ABB RAPID module: Module1.mod

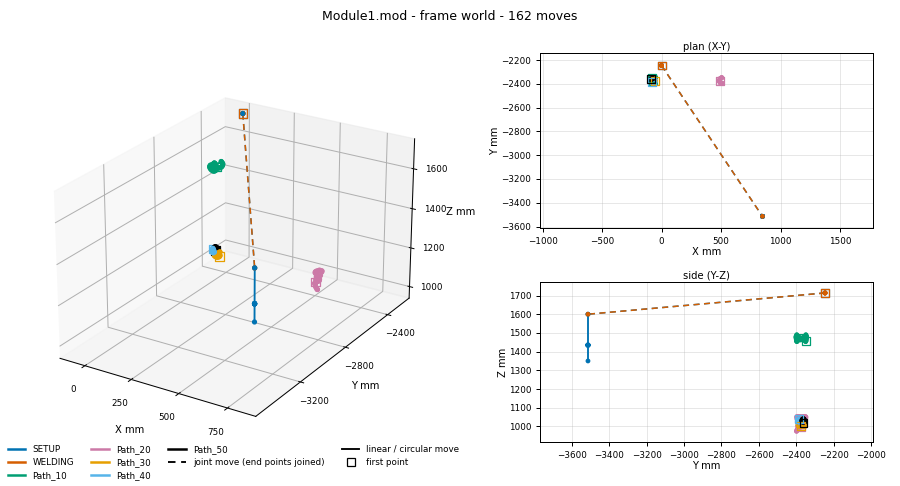
[picture p0: tool path of Module1.mod in frame world, 162 of 162 moves have a stored position in this frame; points joined in program order, loops and branches not executed]
MODULE Module1
    CONST robtarget Target_00:=[[0,-2246.385527781,1713.738524269],[0.23021145,-0.668582596,0.668582596,0.23021145],[0,0,0,0],[9E+09,9E+09,9E+09,9E+09,9E+09,9E+09]];
    CONST robtarget Target_10:=[[-80.421946623,-2349.93093018,1456.191919268],[0.23021145,-0.668582596,0.668582596,0.23021145],[0,0,0,0],[9E+09,9E+09,9E+09,9E+09,9E+09,9E+09]];
    CONST robtarget Target_20:=[[-85.308425352,-2349.8292418,1459.188833121],[0.23021145,-0.668582596,0.668582596,0.23021145],[0,0,0,0],[9E+09,9E+09,9E+09,9E+09,9E+09,9E+09]];
    CONST robtarget Target_30:=[[-89.179888675,-2349.715135272,1463.416236431],[0.23021145,-0.668582596,0.668582596,0.23021145],[0,0,0,0],[9E+09,9E+09,9E+09,9E+09,9E+09,9E+09]];
    CONST robtarget Target_40:=[[-91.78885584,-2349.595757829,1468.705305741],[0.23021145,-0.668582596,0.668582596,0.23021145],[0,0,0,0],[9E+09,9E+09,9E+09,9E+09,9E+09,9E+09]];
    CONST robtarget Target_50:=[[-92.546420184,-2350.235564494,1471.857704903],[0.23021145,-0.668582596,0.668582596,0.23021145],[0,0,0,0],[9E+09,9E+09,9E+09,9E+09,9E+09,9E+09]];
    CONST robtarget Target_60:=[[-92.795669653,-2352.001572523,1474.657635747],[0.23021145,-0.668582596,0.668582596,0.23021145],[0,0,0,0],[9E+09,9E+09,9E+09,9E+09,9E+09,9E+09]];
    CONST robtarget Target_70:=[[-92.744993461,-2354.535100522,1476.584408087],[0.23021145,-0.668582596,0.668582596,0.23021145],[0,0,0,0],[9E+09,9E+09,9E+09,9E+09,9E+09,9E+09]];
    CONST robtarget Target_80:=[[-92.678630412,-2357.601626995,1477.312867316],[0.23021145,-0.668582596,0.668582596,0.23021145],[0,0,0,0],[9E+09,9E+09,9E+09,9E+09,9E+09,9E+09]];
    CONST robtarget Target_10_3:=[[847.938,-3513.969,1435],[0.130526192,0,-0.991444861,0],[-1,0,0,0],[9E+09,9E+09,9E+09,9E+09,9E+09,9E+09]];
    CONST robtarget Target_10_4:=[[847.938,-3513.969,1435],[0.130526192,0,0.991444861,0],[-1,-1,0,0],[9E+09,9E+09,9E+09,9E+09,9E+09,9E+09]];
    CONST robtarget Target_10_2:=[[847.938,-3513.969,1435],[0,0,1,0],[0,-1,0,0],[9E+09,9E+09,9E+09,9E+09,9E+09,9E+09]];
    CONST robtarget Target_10_5:=[[847.938,-3513.969,1435],[0,0,0.991444861,-0.130526192],[-1,-1,0,0],[9E+09,9E+09,9E+09,9E+09,9E+09,9E+09]];
    CONST robtarget Target_10_6:=[[847.938,-3513.969,1435],[0,0,0.991444861,0.130526192],[-2,0,-1,0],[9E+09,9E+09,9E+09,9E+09,9E+09,9E+09]];
    CONST robtarget Target_10_7:=[[847.938,-3513.969,1350],[0,0,1,0],[-1,-1,0,0],[9E+09,9E+09,9E+09,9E+09,9E+09,9E+09]];
    CONST robtarget HOME:=[[0,-2246.385527781,1713.738524269],[0.23021145,-0.668582596,0.668582596,0.23021145],[0,-1,0,0],[9E+09,9E+09,9E+09,9E+09,9E+09,9E+09]];
    CONST robtarget SetUp0:=[[847.938,-3513.969,1600],[0,0,1,0],[0,-1,0,0],[9E+09,9E+09,9E+09,9E+09,9E+09,9E+09]];
    CONST robtarget SetUp1:=[[847.938,-3513.969,1435],[0,0,1,0],[0,-1,0,0],[9E+09,9E+09,9E+09,9E+09,9E+09,9E+09]];
    CONST robtarget SetUp_D:=[[847.938,-3513.969,1435],[0.130526192,0,-0.991444861,0],[-1,0,0,0],[9E+09,9E+09,9E+09,9E+09,9E+09,9E+09]];
    CONST robtarget SetUp_U:=[[847.938,-3513.969,1435],[0.130526192,0,0.991444861,0],[-1,-1,0,0],[9E+09,9E+09,9E+09,9E+09,9E+09,9E+09]];
    CONST robtarget SetUp_L:=[[847.938,-3513.969,1435],[0,0,0.991444861,-0.130526192],[-1,-1,0,0],[9E+09,9E+09,9E+09,9E+09,9E+09,9E+09]];
    CONST robtarget SetUp_R:=[[847.938,-3513.969,1435],[0,0,0.991444861,0.130526192],[-2,0,-1,0],[9E+09,9E+09,9E+09,9E+09,9E+09,9E+09]];
    CONST robtarget SetUp2:=[[847.938,-3513.969,1350],[0,0,1,0],[-1,-1,0,0],[9E+09,9E+09,9E+09,9E+09,9E+09,9E+09]];
    CONST robtarget Target_12:=[[-51.6,-2395.953,1475.08],[0.23021145,-0.668582596,0.668582596,0.23021145],[0,-1,0,0],[9E+09,9E+09,9E+09,9E+09,9E+09,9E+09]];
    CONST robtarget Target_11:=[[-76.443538654,-2395.952996748,1454.921874665],[0.23021145,-0.668582596,0.668582596,0.23021145],[0,-1,0,0],[9E+09,9E+09,9E+09,9E+09,9E+09,9E+09]];
    CONST robtarget Target_13:=[[-58.133756044,-2397.268954021,1490.12991755],[0.23021145,-0.668582596,0.668582596,0.23021145],[0,-1,0,0],[9E+09,9E+09,9E+09,9E+09,9E+09,9E+09]];
    CONST robtarget Target_14:=[[-58.130333404,-2349.245966493,1490.126743663],[0.23021145,-0.668582596,0.668582596,0.23021145],[0,-1,0,0],[9E+09,9E+09,9E+09,9E+09,9E+09,9E+09]];
    CONST robtarget Target_24:=[[-76.443540019,-2395.952934877,1454.921816349],[0.23021145,-0.668582596,0.668582596,0.23021145],[0,0,0,0],[9E+09,9E+09,9E+09,9E+09,9E+09,9E+09]];
    CONST robtarget Target_34:=[[-72.197140196,-2396.852775521,1454.480000199],[0.23021145,-0.668582596,0.668582596,0.23021145],[0,0,0,0],[9E+09,9E+09,9E+09,9E+09,9E+09,9E+09]];
    CONST robtarget Target_44:=[[-68.822373268,-2397.251160157,1454.75878848],[0.23021145,-0.668582596,0.668582596,0.23021145],[0,0,0,0],[9E+09,9E+09,9E+09,9E+09,9E+09,9E+09]];
    CONST robtarget Target_54:=[[-63.419325441,-2398.041235042,1456.445093127],[0.23021145,-0.668582596,0.668582596,0.23021145],[0,0,0,0],[9E+09,9E+09,9E+09,9E+09,9E+09,9E+09]];
    CONST robtarget Target_64:=[[-56.852171112,-2399.35121885,1461.339397818],[0.23021145,-0.668582596,0.668582596,0.23021145],[0,0,0,0],[9E+09,9E+09,9E+09,9E+09,9E+09,9E+09]];
    CONST robtarget Target_74:=[[-52.904973041,-2400.580201887,1467.86460433],[0.23021145,-0.668582596,0.668582596,0.23021145],[0,0,0,0],[9E+09,9E+09,9E+09,9E+09,9E+09,9E+09]];
    CONST robtarget Target_84:=[[-51.602040443,-2401.574973711,1474.790065418],[0.23021145,-0.668582596,0.668582596,0.23021145],[0,0,0,0],[9E+09,9E+09,9E+09,9E+09,9E+09,9E+09]];
    CONST robtarget Target_94:=[[-51.753594032,-2401.880985924,1477.590872953],[0.23021145,-0.668582596,0.668582596,0.23021145],[0,0,0,0],[9E+09,9E+09,9E+09,9E+09,9E+09,9E+09]];
    CONST robtarget Target_104:=[[-52.921425627,-2401.219597479,1482.339240328],[0.23021145,-0.668582596,0.668582596,0.23021145],[0,0,0,0],[9E+09,9E+09,9E+09,9E+09,9E+09,9E+09]];
    CONST robtarget Target_114:=[[-56.936344557,-2398.168943835,1488.914045775],[0.23021145,-0.668582596,0.668582596,0.23021145],[0,0,0,0],[9E+09,9E+09,9E+09,9E+09,9E+09,9E+09]];
    CONST robtarget Target_124:=[[-58.13387415,-2397.086440024,1490.130053275],[0.23021145,-0.668582596,0.668582596,0.23021145],[0,0,0,0],[9E+09,9E+09,9E+09,9E+09,9E+09,9E+09]];
    CONST robtarget Target_134:=[[-58.085063514,-2349.180158559,1490.084284988],[0.23021145,-0.668582596,0.668582596,0.23021145],[0,0,0,0],[9E+09,9E+09,9E+09,9E+09,9E+09,9E+09]];
    CONST robtarget Target_144:=[[-56.934648376,-2348.363913463,1488.91217408],[0.23021145,-0.668582596,0.668582596,0.23021145],[0,0,0,0],[9E+09,9E+09,9E+09,9E+09,9E+09,9E+09]];
    CONST robtarget Target_154:=[[-52.920814209,-2345.314117052,1482.337616361],[0.23021145,-0.668582596,0.668582596,0.23021145],[0,0,0,0],[9E+09,9E+09,9E+09,9E+09,9E+09,9E+09]];
    CONST robtarget Target_164:=[[-51.75346743,-2344.653327795,1477.589841799],[0.23021145,-0.668582596,0.668582596,0.23021145],[0,0,0,0],[9E+09,9E+09,9E+09,9E+09,9E+09,9E+09]];
    CONST robtarget Target_174:=[[-51.602106701,-2344.95991739,1474.785395815],[0.23021145,-0.668582596,0.668582596,0.23021145],[0,0,0,0],[9E+09,9E+09,9E+09,9E+09,9E+09,9E+09]];
    CONST robtarget Target_184:=[[-52.906744673,-2345.954949784,1467.859868499],[0.23021145,-0.668582596,0.668582596,0.23021145],[0,0,0,0],[9E+09,9E+09,9E+09,9E+09,9E+09,9E+09]];
    CONST robtarget Target_194:=[[-56.855846082,-2347.184083727,1461.335294093],[0.23021145,-0.668582596,0.668582596,0.23021145],[0,0,0,0],[9E+09,9E+09,9E+09,9E+09,9E+09,9E+09]];
    CONST robtarget Target_204:=[[-63.424235174,-2348.493945291,1456.442780476],[0.23021145,-0.668582596,0.668582596,0.23021145],[0,0,0,0],[9E+09,9E+09,9E+09,9E+09,9E+09,9E+09]];
    CONST robtarget Target_214:=[[-68.825579531,-2349.283560155,1454.75825582],[0.23021145,-0.668582596,0.668582596,0.23021145],[0,0,0,0],[9E+09,9E+09,9E+09,9E+09,9E+09,9E+09]];
    CONST robtarget Target_224:=[[-72.19902246,-2349.681691113,1454.480000023],[0.23021145,-0.668582596,0.668582596,0.23021145],[0,0,0,0],[9E+09,9E+09,9E+09,9E+09,9E+09,9E+09]];
    CONST robtarget Target_234:=[[-76.44321562,-2350.581156993,1454.921748062],[0.23021145,-0.668582596,0.668582596,0.23021145],[0,0,0,0],[9E+09,9E+09,9E+09,9E+09,9E+09,9E+09]];
    CONST robtarget Target_90:=[[-92.744993461,-2360.668153479,1476.584408087],[0.23021145,-0.668582596,0.668582596,0.23021145],[0,0,0,0],[9E+09,9E+09,9E+09,9E+09,9E+09,9E+09]];
    CONST robtarget Target_100:=[[-92.795669653,-2363.201681499,1474.657635755],[0.23021145,-0.668582596,0.668582596,0.23021145],[0,0,0,0],[9E+09,9E+09,9E+09,9E+09,9E+09,9E+09]];
    CONST robtarget Target_110:=[[-92.546420186,-2364.967689563,1471.857704913],[0.23021145,-0.668582596,0.668582596,0.23021145],[0,0,0,0],[9E+09,9E+09,9E+09,9E+09,9E+09,9E+09]];
    CONST robtarget Target_120:=[[-91.839938652,-2365.605807958,1468.864470277],[0.23021145,-0.668582596,0.668582596,0.23021145],[0,0,0,0],[9E+09,9E+09,9E+09,9E+09,9E+09,9E+09]];
    CONST robtarget Target_130:=[[-89.587784657,-2365.715117705,1464.033509845],[0.23021145,-0.668582596,0.668582596,0.23021145],[0,0,0,0],[9E+09,9E+09,9E+09,9E+09,9E+09,9E+09]];
    CONST robtarget Target_140:=[[-88.012549549,-2365.769448615,1461.876845954],[0.23021145,-0.668582596,0.668582596,0.23021145],[0,0,0,0],[9E+09,9E+09,9E+09,9E+09,9E+09,9E+09]];
    CONST robtarget Target_150:=[[-89.33341612,-2369.703848018,1463.642952652],[0.23021145,-0.668582596,0.668582596,0.23021145],[0,0,0,0],[9E+09,9E+09,9E+09,9E+09,9E+09,9E+09]];
    CONST robtarget Target_160:=[[-89.564284895,-2375.442842076,1463.995789049],[0.23021145,-0.668582596,0.668582596,0.23021145],[0,0,0,0],[9E+09,9E+09,9E+09,9E+09,9E+09,9E+09]];
    CONST robtarget Target_170:=[[-88.012549549,-2380.764551385,1461.876845954],[0.23021145,-0.668582596,0.668582596,0.23021145],[0,0,0,0],[9E+09,9E+09,9E+09,9E+09,9E+09,9E+09]];
    CONST robtarget Target_180:=[[-90.87076908,-2380.873736507,1466.375841111],[0.23021145,-0.668582596,0.668582596,0.23021145],[0,0,0,0],[9E+09,9E+09,9E+09,9E+09,9E+09,9E+09]];
    CONST robtarget Target_190:=[[-91.839938652,-2380.928192042,1468.864470277],[0.23021145,-0.668582596,0.668582596,0.23021145],[0,0,0,0],[9E+09,9E+09,9E+09,9E+09,9E+09,9E+09]];
    CONST robtarget Target_200:=[[-92.546420186,-2381.566310437,1471.857704913],[0.23021145,-0.668582596,0.668582596,0.23021145],[0,0,0,0],[9E+09,9E+09,9E+09,9E+09,9E+09,9E+09]];
    CONST robtarget Target_210:=[[-92.795669653,-2383.332318501,1474.657635755],[0.23021145,-0.668582596,0.668582596,0.23021145],[0,0,0,0],[9E+09,9E+09,9E+09,9E+09,9E+09,9E+09]];
    CONST robtarget Target_220:=[[-92.744993461,-2385.865846521,1476.584408087],[0.23021145,-0.668582596,0.668582596,0.23021145],[0,0,0,0],[9E+09,9E+09,9E+09,9E+09,9E+09,9E+09]];
    CONST robtarget Target_230:=[[-92.678630412,-2388.932373005,1477.312867316],[0.23021145,-0.668582596,0.668582596,0.23021145],[0,0,0,0],[9E+09,9E+09,9E+09,9E+09,9E+09,9E+09]];
    CONST robtarget Target_240:=[[-92.746440422,-2392.039214818,1476.564515404],[0.23021145,-0.668582596,0.668582596,0.23021145],[0,0,0,0],[9E+09,9E+09,9E+09,9E+09,9E+09,9E+09]];
    CONST robtarget Target_250:=[[-92.794171787,-2394.593377395,1474.590011823],[0.23021145,-0.668582596,0.668582596,0.23021145],[0,0,0,0],[9E+09,9E+09,9E+09,9E+09,9E+09,9E+09]];
    CONST robtarget Target_260:=[[-92.539794211,-2396.315236381,1471.816141629],[0.23021145,-0.668582596,0.668582596,0.23021145],[0,0,0,0],[9E+09,9E+09,9E+09,9E+09,9E+09,9E+09]];
    CONST robtarget Target_270:=[[-91.736560317,-2396.936553874,1468.546791677],[0.23021145,-0.668582596,0.668582596,0.23021145],[0,0,0,0],[9E+09,9E+09,9E+09,9E+09,9E+09,9E+09]];
    CONST robtarget Target_280:=[[-89.179888675,-2396.818864728,1463.416236431],[0.23021145,-0.668582596,0.668582596,0.23021145],[0,0,0,0],[9E+09,9E+09,9E+09,9E+09,9E+09,9E+09]];
    CONST robtarget Target_290:=[[-85.308425352,-2396.7047582,1459.188833121],[0.23021145,-0.668582596,0.668582596,0.23021145],[0,0,0,0],[9E+09,9E+09,9E+09,9E+09,9E+09,9E+09]];
    CONST robtarget Target_300:=[[-80.421946623,-2396.60306982,1456.191919268],[0.23021145,-0.668582596,0.668582596,0.23021145],[0,0,0,0],[9E+09,9E+09,9E+09,9E+09,9E+09,9E+09]];
    CONST robtarget Target_310:=[[-76.443540019,-2395.952934877,1454.921816349],[0.23021145,-0.668582596,0.668582596,0.23021145],[0,0,0,0],[9E+09,9E+09,9E+09,9E+09,9E+09,9E+09]];
    CONST robtarget Target_320:=[[-72.197140196,-2396.852775521,1454.480000199],[0.23021145,-0.668582596,0.668582596,0.23021145],[0,0,0,0],[9E+09,9E+09,9E+09,9E+09,9E+09,9E+09]];
    CONST robtarget Target_330:=[[-68.822373268,-2397.251160157,1454.75878848],[0.23021145,-0.668582596,0.668582596,0.23021145],[0,0,0,0],[9E+09,9E+09,9E+09,9E+09,9E+09,9E+09]];
    CONST robtarget Target_340:=[[-63.419325441,-2398.041235042,1456.445093127],[0.23021145,-0.668582596,0.668582596,0.23021145],[0,0,0,0],[9E+09,9E+09,9E+09,9E+09,9E+09,9E+09]];
    CONST robtarget Target_350:=[[-56.852171112,-2399.35121885,1461.339397818],[0.23021145,-0.668582596,0.668582596,0.23021145],[0,0,0,0],[9E+09,9E+09,9E+09,9E+09,9E+09,9E+09]];
    CONST robtarget Target_360:=[[-52.904973041,-2400.580201887,1467.86460433],[0.23021145,-0.668582596,0.668582596,0.23021145],[0,0,0,0],[9E+09,9E+09,9E+09,9E+09,9E+09,9E+09]];
    CONST robtarget Target_370:=[[-51.602040443,-2401.574973711,1474.790065418],[0.23021145,-0.668582596,0.668582596,0.23021145],[0,0,0,0],[9E+09,9E+09,9E+09,9E+09,9E+09,9E+09]];
    CONST robtarget Target_380:=[[-51.753594032,-2401.880985924,1477.590872953],[0.23021145,-0.668582596,0.668582596,0.23021145],[0,0,0,0],[9E+09,9E+09,9E+09,9E+09,9E+09,9E+09]];
    CONST robtarget Target_390:=[[-52.921425627,-2401.219597479,1482.339240328],[0.23021145,-0.668582596,0.668582596,0.23021145],[0,0,0,0],[9E+09,9E+09,9E+09,9E+09,9E+09,9E+09]];
    CONST robtarget Target_400:=[[-56.936344557,-2398.168943835,1488.914045775],[0.23021145,-0.668582596,0.668582596,0.23021145],[0,0,0,0],[9E+09,9E+09,9E+09,9E+09,9E+09,9E+09]];
    CONST robtarget Target_410:=[[-58.13387415,-2397.086440024,1490.130053275],[0.23021145,-0.668582596,0.668582596,0.23021145],[0,0,0,0],[9E+09,9E+09,9E+09,9E+09,9E+09,9E+09]];
    CONST robtarget Target_420:=[[-58.085063514,-2349.180158559,1490.084284988],[0.23021145,-0.668582596,0.668582596,0.23021145],[0,0,0,0],[9E+09,9E+09,9E+09,9E+09,9E+09,9E+09]];
    CONST robtarget Target_430:=[[-56.934648376,-2348.363913463,1488.91217408],[0.23021145,-0.668582596,0.668582596,0.23021145],[0,0,0,0],[9E+09,9E+09,9E+09,9E+09,9E+09,9E+09]];
    CONST robtarget Target_440:=[[-52.920814209,-2345.314117052,1482.337616361],[0.23021145,-0.668582596,0.668582596,0.23021145],[0,0,0,0],[9E+09,9E+09,9E+09,9E+09,9E+09,9E+09]];
    CONST robtarget Target_450:=[[-51.75346743,-2344.653327795,1477.589841799],[0.23021145,-0.668582596,0.668582596,0.23021145],[0,0,0,0],[9E+09,9E+09,9E+09,9E+09,9E+09,9E+09]];
    CONST robtarget Target_460:=[[-51.602106701,-2344.95991739,1474.785395815],[0.23021145,-0.668582596,0.668582596,0.23021145],[0,0,0,0],[9E+09,9E+09,9E+09,9E+09,9E+09,9E+09]];
    CONST robtarget Target_470:=[[-52.906744673,-2345.954949784,1467.859868499],[0.23021145,-0.668582596,0.668582596,0.23021145],[0,0,0,0],[9E+09,9E+09,9E+09,9E+09,9E+09,9E+09]];
    CONST robtarget Target_480:=[[-56.855846082,-2347.184083727,1461.335294093],[0.23021145,-0.668582596,0.668582596,0.23021145],[0,0,0,0],[9E+09,9E+09,9E+09,9E+09,9E+09,9E+09]];
    CONST robtarget Target_490:=[[-63.424235174,-2348.493945291,1456.442780476],[0.23021145,-0.668582596,0.668582596,0.23021145],[0,0,0,0],[9E+09,9E+09,9E+09,9E+09,9E+09,9E+09]];
    CONST robtarget Target_500:=[[-68.825579531,-2349.283560155,1454.75825582],[0.23021145,-0.668582596,0.668582596,0.23021145],[0,0,0,0],[9E+09,9E+09,9E+09,9E+09,9E+09,9E+09]];
    CONST robtarget Target_510:=[[-72.19902246,-2349.681691113,1454.480000023],[0.23021145,-0.668582596,0.668582596,0.23021145],[0,0,0,0],[9E+09,9E+09,9E+09,9E+09,9E+09,9E+09]];
    CONST robtarget Target_520:=[[-76.44321562,-2350.581156993,1454.921748062],[0.23021145,-0.668582596,0.668582596,0.23021145],[0,0,0,0],[9E+09,9E+09,9E+09,9E+09,9E+09,9E+09]];
    CONST robtarget Target_530:=[[487.299996993,-2373.276917925,996.628436583],[0.23021145,-0.668582596,0.668582596,0.23021145],[-1,1,-2,0],[9E+09,9E+09,9E+09,9E+09,9E+09,9E+09]];
    CONST robtarget Target_540:=[[488.426755723,-2365.810441523,996.645880622],[0.23021145,-0.668582596,0.668582596,0.23021145],[-1,1,-2,0],[9E+09,9E+09,9E+09,9E+09,9E+09,9E+09]];
    CONST robtarget Target_550:=[[491.55563648,-2359.233567409,996.708468698],[0.23021145,-0.668582596,0.668582596,0.23021145],[-1,1,-2,0],[9E+09,9E+09,9E+09,9E+09,9E+09,9E+09]];
    CONST robtarget Target_560:=[[494.335480711,-2355.77020944,997.759340006],[0.23021145,-0.668582596,0.668582596,0.23021145],[-1,1,-2,0],[9E+09,9E+09,9E+09,9E+09,9E+09,9E+09]];
    CONST robtarget Target_570:=[[496.045256041,-2354.144982745,999.868648152],[0.23021145,-0.668582596,0.668582596,0.23021145],[-1,1,-2,0],[9E+09,9E+09,9E+09,9E+09,9E+09,9E+09]];
    CONST robtarget Target_580:=[[497.160176535,-2353.235508153,1006.214893507],[0.23021145,-0.668582596,0.668582596,0.23021145],[-1,1,-2,0],[9E+09,9E+09,9E+09,9E+09,9E+09,9E+09]];
    CONST robtarget Target_590:=[[500.454275244,-2351.089179936,1025.568620281],[0.23021145,-0.668582596,0.668582596,0.23021145],[-1,1,-2,0],[9E+09,9E+09,9E+09,9E+09,9E+09,9E+09]];
    CONST robtarget Target_600:=[[505.083274082,-2349.119681802,1043.521763826],[0.23021145,-0.668582596,0.668582596,0.23021145],[-1,1,-2,0],[9E+09,9E+09,9E+09,9E+09,9E+09,9E+09]];
    CONST robtarget Target_610:=[[507.343085984,-2348.529462968,1049.012274976],[0.23021145,-0.668582596,0.668582596,0.23021145],[-1,1,-2,0],[9E+09,9E+09,9E+09,9E+09,9E+09,9E+09]];
    CONST robtarget Target_620:=[[505.535623849,-2348.983594014,1051.461886961],[0.23021145,-0.668582596,0.668582596,0.23021145],[-1,1,-2,0],[9E+09,9E+09,9E+09,9E+09,9E+09,9E+09]];
    CONST robtarget Target_630:=[[497.352082522,-2353.088515517,1053.866566899],[0.23021145,-0.668582596,0.668582596,0.23021145],[-1,1,-2,0],[9E+09,9E+09,9E+09,9E+09,9E+09,9E+09]];
    CONST robtarget Target_640:=[[494.509628643,-2355.589982259,1053.637220967],[0.23021145,-0.668582596,0.668582596,0.23021145],[-1,1,-2,0],[9E+09,9E+09,9E+09,9E+09,9E+09,9E+09]];
    CONST robtarget Target_650:=[[488.667708806,-2365.071097708,1053.144110545],[0.23021145,-0.668582596,0.668582596,0.23021145],[-1,1,-2,0],[9E+09,9E+09,9E+09,9E+09,9E+09,9E+09]];
    CONST robtarget Target_660:=[[487.387269654,-2375.378246342,1053.051278916],[0.23021145,-0.668582596,0.668582596,0.23021145],[-1,1,-2,0],[9E+09,9E+09,9E+09,9E+09,9E+09,9E+09]];
    CONST robtarget Target_670:=[[490.179034965,-2384.99905795,1053.264272624],[0.23021145,-0.668582596,0.668582596,0.23021145],[-1,1,-2,0],[9E+09,9E+09,9E+09,9E+09,9E+09,9E+09]];
    CONST robtarget Target_680:=[[495.944189315,-2392.323329916,1053.761721465],[0.23021145,-0.668582596,0.668582596,0.23021145],[-1,1,-2,0],[9E+09,9E+09,9E+09,9E+09,9E+09,9E+09]];
    CONST robtarget Target_690:=[[501.923570503,-2396.21407252,1053.095408329],[0.23021145,-0.668582596,0.668582596,0.23021145],[-1,1,-2,0],[9E+09,9E+09,9E+09,9E+09,9E+09,9E+09]];
    CONST robtarget Target_700:=[[506.439669165,-2397.815729032,1050.82197549],[0.23021145,-0.668582596,0.668582596,0.23021145],[-1,1,-2,0],[9E+09,9E+09,9E+09,9E+09,9E+09,9E+09]];
    CONST robtarget Target_710:=[[507.144983742,-2397.982212796,1048.566827679],[0.23021145,-0.668582596,0.668582596,0.23021145],[-1,1,-2,0],[9E+09,9E+09,9E+09,9E+09,9E+09,9E+09]];
    CONST robtarget Target_720:=[[503.951891927,-2397.053737866,1040.029521343],[0.23021145,-0.668582596,0.668582596,0.23021145],[-1,1,-2,0],[9E+09,9E+09,9E+09,9E+09,9E+09,9E+09]];
    CONST robtarget Target_730:=[[499.997406812,-2395.216000901,1023.302279311],[0.23021145,-0.668582596,0.668582596,0.23021145],[-1,1,-2,0],[9E+09,9E+09,9E+09,9E+09,9E+09,9E+09]];
    CONST robtarget Target_740:=[[496.479221848,-2392.776252582,1001.364855986],[0.23021145,-0.668582596,0.668582596,0.23021145],[-1,1,-2,0],[9E+09,9E+09,9E+09,9E+09,9E+09,9E+09]];
    CONST robtarget Target_750:=[[495.294214654,-2391.732569093,998.701869528],[0.23021145,-0.668582596,0.668582596,0.23021145],[-1,1,-2,0],[9E+09,9E+09,9E+09,9E+09,9E+09,9E+09]];
    CONST robtarget Target_760:=[[492.470619494,-2388.603755526,996.798168653],[0.23021145,-0.668582596,0.668582596,0.23021145],[-1,1,-2,0],[9E+09,9E+09,9E+09,9E+09,9E+09,9E+09]];
    CONST robtarget Target_770:=[[488.505147517,-2380.992896643,996.6471506],[0.23021145,-0.668582596,0.668582596,0.23021145],[-1,1,-2,0],[9E+09,9E+09,9E+09,9E+09,9E+09,9E+09]];
    CONST robtarget Target_780:=[[487.299996993,-2373.276917925,996.628436583],[0.23021145,-0.668582596,0.668582596,0.23021145],[-1,1,-2,0],[9E+09,9E+09,9E+09,9E+09,9E+09,9E+09]];
    CONST robtarget Target_790:=[[487.981958123,-2379.111828796,995.950630211],[0.23021145,-0.668582596,0.668582596,0.23021145],[-1,1,-2,0],[9E+09,9E+09,9E+09,9E+09,9E+09,9E+09]];
    CONST robtarget Target_800:=[[489.994132771,-2384.637936154,993.953157034],[0.23021145,-0.668582596,0.668582596,0.23021145],[-1,1,-2,0],[9E+09,9E+09,9E+09,9E+09,9E+09,9E+09]];
    CONST robtarget Target_810:=[[495.76754704,-2392.165317816,988.249411952],[0.23021145,-0.668582596,0.668582596,0.23021145],[-1,1,-2,0],[9E+09,9E+09,9E+09,9E+09,9E+09,9E+09]];
    CONST robtarget Target_820:=[[501.496703829,-2396.008877824,982.655438281],[0.23021145,-0.668582596,0.668582596,0.23021145],[-1,1,-2,0],[9E+09,9E+09,9E+09,9E+09,9E+09,9E+09]];
    CONST robtarget Target_830:=[[508.674571782,-2398.270882556,976.137956475],[0.23021145,-0.668582596,0.668582596,0.23021145],[-1,1,-2,0],[9E+09,9E+09,9E+09,9E+09,9E+09,9E+09]];
    CONST robtarget Target_840:=[[511.939956729,-2398.56865142,974.442449041],[0.23021145,-0.668582596,0.668582596,0.23021145],[-1,1,-2,0],[9E+09,9E+09,9E+09,9E+09,9E+09,9E+09]];
    CONST robtarget Target_850:=[[512.599996976,-2398.577262632,974.452581349],[0.23021145,-0.668582596,0.668582596,0.23021145],[-1,1,-2,0],[9E+09,9E+09,9E+09,9E+09,9E+09,9E+09]];
    CONST robtarget Target_860:=[[-54.7,-2373.267,1000.432815492],[0.23021145,-0.668582596,0.668582596,0.23021145],[0,0,-1,1],[9E+09,9E+09,9E+09,9E+09,9E+09,9E+09]];
    CONST robtarget Target_870:=[[-55.380995074,-2378.101363794,1000.496914037],[0.23021145,-0.668582596,0.668582596,0.23021145],[0,0,-1,1],[9E+09,9E+09,9E+09,9E+09,9E+09,9E+09]];
    CONST robtarget Target_880:=[[-57.788499967,-2383.194671771,1000.723520023],[0.23021145,-0.668582596,0.668582596,0.23021145],[0,0,-1,1],[9E+09,9E+09,9E+09,9E+09,9E+09,9E+09]];
    CONST robtarget Target_890:=[[-61.385577124,-2387.025570342,1001.218021936],[0.23021145,-0.668582596,0.668582596,0.23021145],[0,0,-1,1],[9E+09,9E+09,9E+09,9E+09,9E+09,9E+09]];
    CONST robtarget Target_900:=[[-62.471950319,-2387.813994514,1001.590508019],[0.23021145,-0.668582596,0.668582596,0.23021145],[0,0,-1,1],[9E+09,9E+09,9E+09,9E+09,9E+09,9E+09]];
    CONST robtarget Target_910:=[[-68.179859757,-2390.298983808,1004.519536014],[0.23021145,-0.668582596,0.668582596,0.23021145],[0,0,-1,1],[9E+09,9E+09,9E+09,9E+09,9E+09,9E+09]];
    CONST robtarget Target_920:=[[-72.192285645,-2390.7669983,1007.139615096],[0.23021145,-0.668582596,0.668582596,0.23021145],[0,0,-1,1],[9E+09,9E+09,9E+09,9E+09,9E+09,9E+09]];
    CONST robtarget Target_930:=[[-68.270651803,-2390.320158732,1010.93125149],[0.23021145,-0.668582596,0.668582596,0.23021145],[0,0,-1,1],[9E+09,9E+09,9E+09,9E+09,9E+09,9E+09]];
    CONST robtarget Target_940:=[[-61.470642721,-2387.09200967,1017.210994518],[0.23021145,-0.668582596,0.668582596,0.23021145],[0,0,-1,1],[9E+09,9E+09,9E+09,9E+09,9E+09,9E+09]];
    CONST robtarget Target_950:=[[-57.35452451,-2382.533167357,1021.007974151],[0.23021145,-0.668582596,0.668582596,0.23021145],[0,0,-1,1],[9E+09,9E+09,9E+09,9E+09,9E+09,9E+09]];
    CONST robtarget Target_960:=[[-55.272832166,-2377.70783203,1022.927950698],[0.23021145,-0.668582596,0.668582596,0.23021145],[0,0,-1,1],[9E+09,9E+09,9E+09,9E+09,9E+09,9E+09]];
    CONST robtarget Target_970:=[[-54.713195135,-2372.587547558,1023.444625162],[0.23021145,-0.668582596,0.668582596,0.23021145],[0,0,-1,1],[9E+09,9E+09,9E+09,9E+09,9E+09,9E+09]];
    CONST robtarget Target_980:=[[-55.615920962,-2367.6796641,1022.611333928],[0.23021145,-0.668582596,0.668582596,0.23021145],[0,0,-1,1],[9E+09,9E+09,9E+09,9E+09,9E+09,9E+09]];
    CONST robtarget Target_990:=[[-58.110745564,-2362.8870718,1020.308476237],[0.23021145,-0.668582596,0.668582596,0.23021145],[0,0,-1,1],[9E+09,9E+09,9E+09,9E+09,9E+09,9E+09]];
    CONST robtarget Target_1000:=[[-62.836441832,-2358.482759119,1015.947615391],[0.23021145,-0.668582596,0.668582596,0.23021145],[0,0,-1,1],[9E+09,9E+09,9E+09,9E+09,9E+09,9E+09]];
    CONST robtarget Target_1010:=[[-71.360055278,-2355.787168969,1008.057782451],[0.23021145,-0.668582596,0.668582596,0.23021145],[0,0,-1,1],[9E+09,9E+09,9E+09,9E+09,9E+09,9E+09]];
    CONST robtarget Target_1020:=[[-72.097833841,-2355.767298229,1006.943809206],[0.23021145,-0.668582596,0.668582596,0.23021145],[0,0,-1,1],[9E+09,9E+09,9E+09,9E+09,9E+09,9E+09]];
    CONST robtarget Target_1030:=[[-66.677000111,-2356.661384316,1003.657261773],[0.23021145,-0.668582596,0.668582596,0.23021145],[0,0,-1,1],[9E+09,9E+09,9E+09,9E+09,9E+09,9E+09]];
    CONST robtarget Target_1040:=[[-61.703642001,-2359.264269239,1001.345628088],[0.23021145,-0.668582596,0.668582596,0.23021145],[0,0,-1,1],[9E+09,9E+09,9E+09,9E+09,9E+09,9E+09]];
    CONST robtarget Target_1050:=[[-60.09647453,-2360.627590552,1000.990812213],[0.23021145,-0.668582596,0.668582596,0.23021145],[0,0,-1,1],[9E+09,9E+09,9E+09,9E+09,9E+09,9E+09]];
    CONST robtarget Target_1060:=[[-57.133559565,-2364.364619834,1000.66187387],[0.23021145,-0.668582596,0.668582596,0.23021145],[0,0,-1,1],[9E+09,9E+09,9E+09,9E+09,9E+09,9E+09]];
    CONST robtarget Target_1070:=[[-83.701391589,-2386.456692624,1040.564001432],[0.23021145,-0.668582596,0.668582596,0.23021145],[0,0,-1,1],[9E+09,9E+09,9E+09,9E+09,9E+09,9E+09]];
    CONST robtarget Target_1080:=[[-87.15651289,-2382.352646078,1040.669440907],[0.23021145,-0.668582596,0.668582596,0.23021145],[0,0,-1,1],[9E+09,9E+09,9E+09,9E+09,9E+09,9E+09]];
    CONST robtarget Target_1090:=[[-88.941057524,-2378.364127048,1037.258284446],[0.23021145,-0.668582596,0.668582596,0.23021145],[0,0,-1,1],[9E+09,9E+09,9E+09,9E+09,9E+09,9E+09]];
    CONST robtarget Target_1100:=[[-89.475084515,-2376.06963048,1032.080212204],[0.23021145,-0.668582596,0.668582596,0.23021145],[0,0,-1,1],[9E+09,9E+09,9E+09,9E+09,9E+09,9E+09]];
    CONST robtarget Target_1110:=[[-89.374584474,-2376.626114193,1026.579622599],[0.23021145,-0.668582596,0.668582596,0.23021145],[0,0,-1,1],[9E+09,9E+09,9E+09,9E+09,9E+09,9E+09]];
    CONST robtarget Target_1120:=[[-88.823918204,-2378.734663444,1023.636801699],[0.23021145,-0.668582596,0.668582596,0.23021145],[0,0,-1,1],[9E+09,9E+09,9E+09,9E+09,9E+09,9E+09]];
    CONST robtarget Target_1130:=[[-87.184170591,-2382.307167681,1021.50414475],[0.23021145,-0.668582596,0.668582596,0.23021145],[0,0,-1,1],[9E+09,9E+09,9E+09,9E+09,9E+09,9E+09]];
    CONST robtarget Target_1140:=[[-85.125321065,-2385.064714837,1020.381003904],[0.23021145,-0.668582596,0.668582596,0.23021145],[0,0,-1,1],[9E+09,9E+09,9E+09,9E+09,9E+09,9E+09]];
    CONST robtarget Target_1150:=[[-83.125050807,-2386.937891151,1019.753704124],[0.23021145,-0.668582596,0.668582596,0.23021145],[0,0,-1,1],[9E+09,9E+09,9E+09,9E+09,9E+09,9E+09]];
    CONST robtarget Target_1160:=[[-79.965278406,-2388.949807506,1019.978731251],[0.23021145,-0.668582596,0.668582596,0.23021145],[0,0,-1,1],[9E+09,9E+09,9E+09,9E+09,9E+09,9E+09]];
    CONST robtarget Target_1170:=[[-76.698742788,-2390.178869008,1021.361989514],[0.23021145,-0.668582596,0.668582596,0.23021145],[0,0,-1,1],[9E+09,9E+09,9E+09,9E+09,9E+09,9E+09]];
    CONST robtarget Target_1180:=[[-74.058808637,-2390.668000847,1023.880062652],[0.23021145,-0.668582596,0.668582596,0.23021145],[0,0,-1,1],[9E+09,9E+09,9E+09,9E+09,9E+09,9E+09]];
    CONST robtarget Target_1190:=[[-73.290624881,-2390.73298229,1025.553481425],[0.23021145,-0.668582596,0.668582596,0.23021145],[0,0,-1,1],[9E+09,9E+09,9E+09,9E+09,9E+09,9E+09]];
    CONST robtarget Target_1200:=[[-73.042123166,-2390.746726216,1027.352744546],[0.23021145,-0.668582596,0.668582596,0.23021145],[0,0,-1,1],[9E+09,9E+09,9E+09,9E+09,9E+09,9E+09]];
    CONST robtarget Target_1210:=[[-74.223288825,-2390.649643709,1031.818924146],[0.23021145,-0.668582596,0.668582596,0.23021145],[0,0,-1,1],[9E+09,9E+09,9E+09,9E+09,9E+09,9E+09]];
    CONST robtarget Target_1220:=[[-76.85286346,-2390.137117416,1035.704334782],[0.23021145,-0.668582596,0.668582596,0.23021145],[0,0,-1,1],[9E+09,9E+09,9E+09,9E+09,9E+09,9E+09]];
    CONST robtarget Target_1230:=[[-80.762646715,-2388.529079847,1038.960861249],[0.23021145,-0.668582596,0.668582596,0.23021145],[0,0,-1,1],[9E+09,9E+09,9E+09,9E+09,9E+09,9E+09]];
    CONST robtarget Target_1240:=[[-85.125321065,-2361.469285163,1020.381003904],[0.23021145,-0.668582596,0.668582596,0.23021145],[0,0,-1,1],[9E+09,9E+09,9E+09,9E+09,9E+09,9E+09]];
    CONST robtarget Target_1250:=[[-83.125050807,-2359.596108849,1019.753704124],[0.23021145,-0.668582596,0.668582596,0.23021145],[0,0,-1,1],[9E+09,9E+09,9E+09,9E+09,9E+09,9E+09]];
    CONST robtarget Target_1260:=[[-79.965278406,-2357.584192494,1019.978731251],[0.23021145,-0.668582596,0.668582596,0.23021145],[0,0,-1,1],[9E+09,9E+09,9E+09,9E+09,9E+09,9E+09]];
    CONST robtarget Target_1270:=[[-76.698742788,-2356.355130992,1021.361989514],[0.23021145,-0.668582596,0.668582596,0.23021145],[0,0,-1,1],[9E+09,9E+09,9E+09,9E+09,9E+09,9E+09]];
    CONST robtarget Target_1280:=[[-74.058808637,-2355.865999153,1023.880062652],[0.23021145,-0.668582596,0.668582596,0.23021145],[0,0,-1,1],[9E+09,9E+09,9E+09,9E+09,9E+09,9E+09]];
    CONST robtarget Target_1290:=[[-73.290624881,-2355.80101771,1025.553481425],[0.23021145,-0.668582596,0.668582596,0.23021145],[0,0,-1,1],[9E+09,9E+09,9E+09,9E+09,9E+09,9E+09]];
    CONST robtarget Target_1300:=[[-75.091790027,-2356.008770168,1033.359119774],[0.23021145,-0.668582596,0.668582596,0.23021145],[0,0,-1,1],[9E+09,9E+09,9E+09,9E+09,9E+09,9E+09]];
    CONST robtarget Target_1310:=[[-80.762646715,-2358.004920153,1038.960861249],[0.23021145,-0.668582596,0.668582596,0.23021145],[0,0,-1,1],[9E+09,9E+09,9E+09,9E+09,9E+09,9E+09]];
    CONST robtarget Target_1320:=[[-83.701391589,-2360.077307376,1040.564001432],[0.23021145,-0.668582596,0.668582596,0.23021145],[0,0,-1,1],[9E+09,9E+09,9E+09,9E+09,9E+09,9E+09]];
    CONST robtarget Target_1330:=[[-85.609294174,-2362.022408867,1041.140912922],[0.23021145,-0.668582596,0.668582596,0.23021145],[0,0,-1,1],[9E+09,9E+09,9E+09,9E+09,9E+09,9E+09]];
    CONST robtarget Target_1340:=[[-86.728587665,-2363.511481538,1040.919842202],[0.23021145,-0.668582596,0.668582596,0.23021145],[0,0,-1,1],[9E+09,9E+09,9E+09,9E+09,9E+09,9E+09]];
    CONST robtarget Target_1350:=[[-87.647796435,-2365.04413035,1040.218421385],[0.23021145,-0.668582596,0.668582596,0.23021145],[0,0,-1,1],[9E+09,9E+09,9E+09,9E+09,9E+09,9E+09]];
    CONST robtarget Target_1360:=[[-88.814716109,-2367.77143737,1037.775574053],[0.23021145,-0.668582596,0.668582596,0.23021145],[0,0,-1,1],[9E+09,9E+09,9E+09,9E+09,9E+09,9E+09]];
    CONST robtarget Target_1370:=[[-89.362410478,-2369.846230117,1034.217677389],[0.23021145,-0.668582596,0.668582596,0.23021145],[0,0,-1,1],[9E+09,9E+09,9E+09,9E+09,9E+09,9E+09]];
    CONST robtarget Target_1380:=[[-89.503287088,-2370.650464896,1030.165693084],[0.23021145,-0.668582596,0.668582596,0.23021145],[0,0,-1,1],[9E+09,9E+09,9E+09,9E+09,9E+09,9E+09]];
    CONST robtarget Target_1390:=[[-89.374584474,-2369.907885807,1026.579622599],[0.23021145,-0.668582596,0.668582596,0.23021145],[0,0,-1,1],[9E+09,9E+09,9E+09,9E+09,9E+09,9E+09]];
    CONST robtarget Target_1400:=[[-88.823918204,-2367.799336556,1023.636801699],[0.23021145,-0.668582596,0.668582596,0.23021145],[0,0,-1,1],[9E+09,9E+09,9E+09,9E+09,9E+09,9E+09]];
    CONST robtarget Target_1410:=[[-87.184170591,-2364.226832319,1021.50414475],[0.23021145,-0.668582596,0.668582596,0.23021145],[0,0,-1,1],[9E+09,9E+09,9E+09,9E+09,9E+09,9E+09]];

    PERS bool START1;
    PERS bool STOP1;
    PERS intnum POS;

    !***********************************************************
    !
    ! Módulo:  Module1
    !
    ! Descripción:
    !   <Introduzca la descripción aquí>
    !
    ! Autor: John Panche
    !
    ! Versión: 1.0
    !
    !***********************************************************


    !***********************************************************
    !
    ! Procedimiento Main
    !
    !   Este es el punto de entrada de su programa
    !
    !***********************************************************
    PROC main()
        SETUP;
        WaitDO OUTPUT1,1;
        WaitTime(4);
        WELDING;
        WaitTime(1);
        Set OUTPUT2;
        Reset OUTPUT2;
    ENDPROC
    PROC SETUP()
        MoveJ HOME,v1000,fine,tWeldGun\WObj:=wobj0;
        MoveJ SetUp0,v1000,fine,tWeldGun\WObj:=wobj0;
        MoveL SetUp1,v100,fine,tWeldGun\WObj:=wobj0;
        MoveL SetUp_D,v5,fine,tWeldGun\WObj:=wobj0;
        MoveL SetUp_U,v5,fine,tWeldGun\WObj:=wobj0;
        MoveL SetUp_D,v5,fine,tWeldGun\WObj:=wobj0;
        MoveL SetUp_U,v5,fine,tWeldGun\WObj:=wobj0;
        MoveL SetUp1,v5,fine,tWeldGun\WObj:=wobj0;
        MoveL SetUp_L,v5,fine,tWeldGun\WObj:=wobj0;
        MoveL SetUp_R,v5,fine,tWeldGun\WObj:=wobj0;
        MoveL SetUp_L,v5,fine,tWeldGun\WObj:=wobj0;
        MoveL SetUp_R,v5,fine,tWeldGun\WObj:=wobj0;
        MoveL SetUp1,v5,fine,tWeldGun\WObj:=wobj0;
        MoveL SetUp2,v100,fine,tWeldGun\WObj:=wobj0;
        WaitTime 1;
        MoveL SetUp0,v100,fine,tWeldGun\WObj:=wobj0;
    ENDPROC
    PROC WELDING()
        MoveJ HOME,v1000,fine,tWeldGun\WObj:=wobj0;
        Path_10;
        MoveJ HOME,v1000,fine,tWeldGun\WObj:=wobj0;
        Path_20;
        MoveJ HOME,v1000,fine,tWeldGun\WObj:=wobj0;
        Path_10;
        MoveJ HOME,v1000,fine,tWeldGun\WObj:=wobj0;
        Path_20;
        MoveJ HOME,v1000,fine,tWeldGun\WObj:=wobj0;
        MoveJ SetUp0,v1000,fine,tWeldGun\WObj:=wobj0;
    ENDPROC
    PROC Path_10()
        MoveL Target_10,v1000,fine,tWeldGun\WObj:=wobj0;
        MoveL Target_20,v50,fine,tWeldGun\WObj:=wobj0;
        MoveL Target_30,v50,fine,tWeldGun\WObj:=wobj0;
        MoveL Target_40,v50,fine,tWeldGun\WObj:=wobj0;
        MoveL Target_50,v50,fine,tWeldGun\WObj:=wobj0;
        MoveL Target_60,v50,fine,tWeldGun\WObj:=wobj0;
        MoveL Target_70,v50,fine,tWeldGun\WObj:=wobj0;
        MoveL Target_80,v50,fine,tWeldGun\WObj:=wobj0;
        MoveL Target_90,v50,fine,tWeldGun\WObj:=wobj0;
        MoveL Target_100,v50,fine,tWeldGun\WObj:=wobj0;
        MoveL Target_110,v50,fine,tWeldGun\WObj:=wobj0;
        MoveL Target_120,v50,fine,tWeldGun\WObj:=wobj0;
        MoveL Target_130,v50,fine,tWeldGun\WObj:=wobj0;
        MoveL Target_140,v50,fine,tWeldGun\WObj:=wobj0;
        MoveL Target_150,v50,fine,tWeldGun\WObj:=wobj0;
        MoveL Target_160,v50,fine,tWeldGun\WObj:=wobj0;
        MoveL Target_170,v50,fine,tWeldGun\WObj:=wobj0;
        MoveL Target_180,v50,fine,tWeldGun\WObj:=wobj0;
        MoveL Target_190,v50,fine,tWeldGun\WObj:=wobj0;
        MoveL Target_200,v50,fine,tWeldGun\WObj:=wobj0;
        MoveL Target_210,v50,fine,tWeldGun\WObj:=wobj0;
        MoveL Target_220,v50,fine,tWeldGun\WObj:=wobj0;
        MoveL Target_230,v50,fine,tWeldGun\WObj:=wobj0;
        MoveL Target_240,v50,fine,tWeldGun\WObj:=wobj0;
        MoveL Target_250,v50,fine,tWeldGun\WObj:=wobj0;
        MoveL Target_260,v50,fine,tWeldGun\WObj:=wobj0;
        MoveL Target_270,v50,fine,tWeldGun\WObj:=wobj0;
        MoveL Target_280,v50,fine,tWeldGun\WObj:=wobj0;
        MoveL Target_290,v50,fine,tWeldGun\WObj:=wobj0;
        MoveL Target_300,v50,fine,tWeldGun\WObj:=wobj0;
        MoveL Target_310,v50,fine,tWeldGun\WObj:=wobj0;
        MoveL Target_320,v50,fine,tWeldGun\WObj:=wobj0;
        MoveL Target_330,v50,fine,tWeldGun\WObj:=wobj0;
        MoveL Target_340,v50,fine,tWeldGun\WObj:=wobj0;
        MoveL Target_350,v50,fine,tWeldGun\WObj:=wobj0;
        MoveL Target_360,v50,fine,tWeldGun\WObj:=wobj0;
        MoveL Target_370,v50,fine,tWeldGun\WObj:=wobj0;
        MoveL Target_380,v50,fine,tWeldGun\WObj:=wobj0;
        MoveL Target_390,v50,fine,tWeldGun\WObj:=wobj0;
        MoveL Target_400,v50,fine,tWeldGun\WObj:=wobj0;
        MoveL Target_410,v50,fine,tWeldGun\WObj:=wobj0;
        MoveL Target_420,v50,fine,tWeldGun\WObj:=wobj0;
        MoveL Target_430,v50,fine,tWeldGun\WObj:=wobj0;
        MoveL Target_440,v50,fine,tWeldGun\WObj:=wobj0;
        MoveL Target_450,v50,fine,tWeldGun\WObj:=wobj0;
        MoveL Target_460,v50,fine,tWeldGun\WObj:=wobj0;
        MoveL Target_470,v50,fine,tWeldGun\WObj:=wobj0;
        MoveL Target_480,v50,fine,tWeldGun\WObj:=wobj0;
        MoveL Target_490,v50,fine,tWeldGun\WObj:=wobj0;
        MoveL Target_500,v50,fine,tWeldGun\WObj:=wobj0;
        MoveL Target_510,v50,fine,tWeldGun\WObj:=wobj0;
        MoveL Target_520,v50,fine,tWeldGun\WObj:=wobj0;
    ENDPROC
    PROC Path_20()
        MoveL Target_530,v1000,fine,tWeldGun\WObj:=wobj0;
        MoveL Target_540,v50,fine,tWeldGun\WObj:=wobj0;
        MoveL Target_550,v50,fine,tWeldGun\WObj:=wobj0;
        MoveL Target_560,v50,fine,tWeldGun\WObj:=wobj0;
        MoveL Target_570,v50,fine,tWeldGun\WObj:=wobj0;
        MoveL Target_580,v50,fine,tWeldGun\WObj:=wobj0;
        MoveL Target_590,v50,fine,tWeldGun\WObj:=wobj0;
        MoveL Target_600,v50,fine,tWeldGun\WObj:=wobj0;
        MoveL Target_610,v50,fine,tWeldGun\WObj:=wobj0;
        MoveL Target_620,v50,fine,tWeldGun\WObj:=wobj0;
        MoveL Target_630,v50,fine,tWeldGun\WObj:=wobj0;
        MoveL Target_640,v50,fine,tWeldGun\WObj:=wobj0;
        MoveL Target_650,v50,fine,tWeldGun\WObj:=wobj0;
        MoveL Target_660,v50,fine,tWeldGun\WObj:=wobj0;
        MoveL Target_670,v50,fine,tWeldGun\WObj:=wobj0;
        MoveL Target_680,v50,fine,tWeldGun\WObj:=wobj0;
        MoveL Target_690,v50,fine,tWeldGun\WObj:=wobj0;
        MoveL Target_700,v50,fine,tWeldGun\WObj:=wobj0;
        MoveL Target_710,v50,fine,tWeldGun\WObj:=wobj0;
        MoveL Target_720,v50,fine,tWeldGun\WObj:=wobj0;
        MoveL Target_730,v50,fine,tWeldGun\WObj:=wobj0;
        MoveL Target_740,v50,fine,tWeldGun\WObj:=wobj0;
        MoveL Target_750,v50,fine,tWeldGun\WObj:=wobj0;
        MoveL Target_760,v50,fine,tWeldGun\WObj:=wobj0;
        MoveL Target_770,v50,fine,tWeldGun\WObj:=wobj0;
        MoveL Target_780,v50,fine,tWeldGun\WObj:=wobj0;
        MoveL Target_790,v50,fine,tWeldGun\WObj:=wobj0;
        MoveL Target_800,v50,fine,tWeldGun\WObj:=wobj0;
        MoveL Target_810,v50,fine,tWeldGun\WObj:=wobj0;
        MoveL Target_820,v50,fine,tWeldGun\WObj:=wobj0;
        MoveL Target_830,v50,fine,tWeldGun\WObj:=wobj0;
        MoveL Target_840,v50,fine,tWeldGun\WObj:=wobj0;
        MoveL Target_850,v50,fine,tWeldGun\WObj:=wobj0;
    ENDPROC
    PROC Path_30()
        MoveL Target_860,v1000,fine,tWeldGun\WObj:=wobj0;
        MoveL Target_870,v5,fine,tWeldGun\WObj:=wobj0;
        MoveL Target_880,v5,fine,tWeldGun\WObj:=wobj0;
        MoveL Target_890,v5,fine,tWeldGun\WObj:=wobj0;
        MoveL Target_900,v5,fine,tWeldGun\WObj:=wobj0;
        MoveL Target_910,v5,fine,tWeldGun\WObj:=wobj0;
        MoveL Target_920,v5,fine,tWeldGun\WObj:=wobj0;
        MoveL Target_930,v5,fine,tWeldGun\WObj:=wobj0;
        MoveL Target_940,v5,fine,tWeldGun\WObj:=wobj0;
        MoveL Target_950,v5,fine,tWeldGun\WObj:=wobj0;
        MoveL Target_960,v5,fine,tWeldGun\WObj:=wobj0;
        MoveL Target_970,v5,fine,tWeldGun\WObj:=wobj0;
        MoveL Target_980,v5,fine,tWeldGun\WObj:=wobj0;
        MoveL Target_990,v5,fine,tWeldGun\WObj:=wobj0;
        MoveL Target_1000,v5,fine,tWeldGun\WObj:=wobj0;
        MoveL Target_1010,v5,fine,tWeldGun\WObj:=wobj0;
        MoveL Target_1020,v5,fine,tWeldGun\WObj:=wobj0;
        MoveL Target_1030,v5,fine,tWeldGun\WObj:=wobj0;
        MoveL Target_1040,v5,fine,tWeldGun\WObj:=wobj0;
        MoveL Target_1050,v5,fine,tWeldGun\WObj:=wobj0;
        MoveL Target_1060,v5,fine,tWeldGun\WObj:=wobj0;
    ENDPROC
    PROC Path_40()
        MoveL Target_1070,v1000,fine,tWeldGun\WObj:=wobj0;
        MoveL Target_1080,v5,fine,tWeldGun\WObj:=wobj0;
        MoveL Target_1090,v5,fine,tWeldGun\WObj:=wobj0;
        MoveL Target_1100,v5,fine,tWeldGun\WObj:=wobj0;
        MoveL Target_1110,v5,fine,tWeldGun\WObj:=wobj0;
        MoveL Target_1120,v5,fine,tWeldGun\WObj:=wobj0;
        MoveL Target_1130,v5,fine,tWeldGun\WObj:=wobj0;
        MoveL Target_1140,v5,fine,tWeldGun\WObj:=wobj0;
        MoveL Target_1150,v5,fine,tWeldGun\WObj:=wobj0;
        MoveL Target_1160,v5,fine,tWeldGun\WObj:=wobj0;
        MoveL Target_1170,v5,fine,tWeldGun\WObj:=wobj0;
        MoveL Target_1180,v5,fine,tWeldGun\WObj:=wobj0;
        MoveL Target_1190,v5,fine,tWeldGun\WObj:=wobj0;
        MoveL Target_1200,v5,fine,tWeldGun\WObj:=wobj0;
        MoveL Target_1210,v5,fine,tWeldGun\WObj:=wobj0;
        MoveL Target_1220,v5,fine,tWeldGun\WObj:=wobj0;
        MoveL Target_1230,v5,fine,tWeldGun\WObj:=wobj0;
    ENDPROC
    PROC Path_50()
        MoveL Target_1240,v1000,fine,tWeldGun\WObj:=wobj0;
        MoveL Target_1250,v5,fine,tWeldGun\WObj:=wobj0;
        MoveL Target_1260,v5,fine,tWeldGun\WObj:=wobj0;
        MoveL Target_1270,v5,fine,tWeldGun\WObj:=wobj0;
        MoveL Target_1280,v5,fine,tWeldGun\WObj:=wobj0;
        MoveL Target_1290,v5,fine,tWeldGun\WObj:=wobj0;
        MoveL Target_1300,v5,fine,tWeldGun\WObj:=wobj0;
        MoveL Target_1310,v5,fine,tWeldGun\WObj:=wobj0;
        MoveL Target_1320,v5,fine,tWeldGun\WObj:=wobj0;
        MoveL Target_1330,v5,fine,tWeldGun\WObj:=wobj0;
        MoveL Target_1340,v5,fine,tWeldGun\WObj:=wobj0;
        MoveL Target_1350,v5,fine,tWeldGun\WObj:=wobj0;
        MoveL Target_1360,v5,fine,tWeldGun\WObj:=wobj0;
        MoveL Target_1370,v5,fine,tWeldGun\WObj:=wobj0;
        MoveL Target_1380,v5,fine,tWeldGun\WObj:=wobj0;
        MoveL Target_1390,v5,fine,tWeldGun\WObj:=wobj0;
        MoveL Target_1400,v5,fine,tWeldGun\WObj:=wobj0;
        MoveL Target_1410,v5,fine,tWeldGun\WObj:=wobj0;
    ENDPROC
ENDMODULE
